{attribute addProperty BoxType "KL2702"}
{attribute addProperty Id "Channel_1Channel_E75BD82E00Channel_2Channel_E75BD82E00"}
{attribute addProperty CRC "1288439370"}
{attribute addProperty SizeInBites "0"}
{attribute addProperty SizeInBytes "0"}
TYPE KL2702_4CCC064A :
STRUCT
	{attribute addProperty Name "Channel_1"}
	Channel_1 : Channel_E75BD82E;
	{attribute addProperty Name "Channel_2"}
	Channel_2 : Channel_E75BD82E;
END_STRUCT
END_TYPE

(* stored: Version 1.2.0.0, ProductVersion 3.1.4024.9
   DUT KL2702_4CCC064A: Id {c2032441-02ba-4ca2-ace4-54aa80ddc5d5} *)
